// TIA Portal project "ConveyorBelt (extra)" (V13)

(* hardware
DEVICE "S7300/ET200M-Station_1"  S7-300 station
   slot 0: "Profilschiene_0"  Rail  6ES7 390-1***0-0AA0
   slot 1: "PS 307 5A_1"  PS 307 5A  6ES7 307-1EA00-0AA0
   slot 2: "SIMATIC S7-300"  CPU 314C-2 PN/DP  6ES7 314-6EH04-0AB0  V3.3
      slot 2: "PROFINET-Schnittstelle_1"  PN-IO
         slot 1: "Port_1"  Port
         slot 2: "Port_2"  Port
      slot 5: "DI 24/DO 16_1"  DI24/DO16
      slot 6: "AI 5/AO 2_1"  AI5/AO2
      slot 7: "Zählen_1"  Counter
      slot 8: "Positionieren_1"  Positioning
*)

// ===== PLC "SIMATIC S7-300"  CPU 314C-2 PN/DP =====

VAR_GLOBAL   // PLC tag table "Standard-Variablentabelle"
   "Ix_1S1" AT %I124.0 : Bool;   // Start-Taster (NO)
   "Ix_2S1" AT %I124.1 : Bool;   // Halt-Taster (NC)
   "Ix_3S1" AT %I124.2 : Bool;   // Richten-Taster (NO)
   "Ix_1B1" AT %I124.3 : Bool;   // Werkstück in Werkstückaufnahme (Ausgangsposition)
   "Ix_2B1" AT %I124.4 : Bool;   // Schwenkarm 1, Position Förderband
   "Ix_2B2" AT %I124.5 : Bool;   // Schwenkarm 1, Position Werkstückaufnahme
   "Ix_3B1" AT %I124.6 : Bool;   // Werkstück am Förderbandende
   "Ix_4B1" AT %I124.7 : Bool;   // Hubeinrichtung, Position oben
   "Ix_5B1" AT %I125.1 : Bool;   // Schwenkarm 2, Position Förderband
   "Ix_5B2" AT %I125.2 : Bool;   // Schwenkarm 2, Position Schlitten
   "Ix_6B1" AT %I125.3 : Bool;   // Werkstück in Werkstückaufnahme des Schlittens
   "Ix_7B2" AT %I125.4 : Bool;   // Schlitten, Position Werkstückaufnahme
   "Ix_7B1" AT %I125.5 : Bool;   // Schlitten, Position Werkstückübergabe
   "Ix_8B1" AT %I125.6 : Bool;   // Schwenkarm 3, Position Rollenband
   "Ix_8B2" AT %I125.7 : Bool;   // Schwenkarm 3, Position Schlitten
   "Ix_9B1" AT %I126.0 : Bool;   // Vakuum Greifer 1 eingeschaltet
   "Ix_9B2" AT %I126.1 : Bool;   // Vakuum Greifer 2 eingeschaltet
   "Ix_4B2" AT %I125.0 : Bool;   // Hubeinrichtung, Position unten
   "Ix_9B3" AT %I126.2 : Bool;   // Vakuum Greifer 3 eingeschaltet
   "Qx_1M1" AT %Q124.0 : Bool;   // Schwenkarm 1 zum Transportgut
   "Qx_2M1" AT %Q124.1 : Bool;   // Förderbandantrieb Schub 1 (NC)
   "Qx_2M2" AT %Q124.2 : Bool;   // Förderbandantrieb Schub 2 (NO)
   "Qx_3M1" AT %Q124.3 : Bool;   // Hubeinrichtung nach unten
   "Qx_4M1" AT %Q124.4 : Bool;   // Schwenkarm 2 vom Förderband zum Schlitten
   "Qx_5M1" AT %Q124.5 : Bool;   // Schlitten zum Schwenkarm 2
   "Qx_6M1" AT %Q124.6 : Bool;   // Schwenkarm 3 von der Rollenbahn zum Schlitten
   "Qx_7M1" AT %Q125.2 : Bool;   // Greifer 1 einschalten
   "Qx_7M2" AT %Q124.7 : Bool;   // Greifer 1 ausschalten
   "Qx_7M3" AT %Q125.3 : Bool;   // Greifer 2 einschalten
   "Qx_7M4" AT %Q125.0 : Bool;   // Greifer 2 ausschalten
   "Qx_7M5" AT %Q125.4 : Bool;   // Greifer 3 einschalten
   "Qx_7M6" AT %Q125.1 : Bool;   // Greifer 3 ausschalten
   "Qx_PStart" AT %Q125.5 : Bool;   // Startlampe (grün)
   "Qx_PHalt" AT %Q125.6 : Bool;   // Haltlampe (rot)
   "Qx_PRichten" AT %Q125.7 : Bool;   // Richtenlampe (orange)
   "Mx_Step0" AT %M0.0 : Bool;   // Merker: Step 0
   "Mx_Step1" AT %M0.1 : Bool;   // Merker: Step 1
   "Mx_Step2" AT %M0.2 : Bool;   // Merker: Step 2
   "Mx_Step3" AT %M0.3 : Bool;   // Merker: Step 3
   "Mx_Step4" AT %M0.4 : Bool;   // Merker: Step 4
   "Mx_Step5" AT %M0.5 : Bool;   // Merker: Step 5
   "Mx_Step6a" AT %M0.6 : Bool;   // Merker: Step 6a
   "Mx_Step7" AT %M0.7 : Bool;   // Merker: Step 7
   "Mx_Step8" AT %M1.0 : Bool;   // Merker: Step 8
   "Mx_Step9" AT %M1.1 : Bool;   // Merker: Step 9
   "Mx_Step10" AT %M1.2 : Bool;   // Merker: Step 10
   "Mx_Step11" AT %M1.3 : Bool;   // Merker: Step 11
   "Mx_Step12" AT %M1.4 : Bool;   // Merker: Step 12
   "Mx_Step13" AT %M1.5 : Bool;   // Merker: Step 13
   "Mx_Step14" AT %M1.6 : Bool;   // Merker: Step 14
   "Mx_Step15" AT %M1.7 : Bool;   // Merker: Step 15
   "Mx_Step16" AT %M2.0 : Bool;   // Merker: Step 16
   "Mx_Step17" AT %M2.1 : Bool;   // Merker: Step 17
   "Mx_Step18" AT %M2.2 : Bool;   // Merker: Step 18
   "Mx_Step19" AT %M2.3 : Bool;   // Merker: Step 19
   "Mx_Step20" AT %M2.4 : Bool;   // Merker: Step 20
   "Mx_Step21" AT %M2.5 : Bool;   // Merker: Step 21
   "Mx_Step22" AT %M2.6 : Bool;   // Merker: Step 22
   "Mx_Step23" AT %M2.7 : Bool;   // Merker: Step 23
   "MD0" AT %MD0 : DWord;   // Merker Doppel Wort 0
   "Mx_InitialFlag" AT %M3.0 : Bool;   // Merker: Initialisierung
   "Mx_Ausgangstellung" AT %M10.0 : Bool;   // Merker: Ausgangstellung
   "Mx_InitSchwenkarm1" AT %M10.1 : Bool;   // Merker: Initalisierung Schwenkarm 1
   "Mx_InitSchwenkarm2" AT %M10.2 : Bool;
   "Mx_InitHubeinrichtung" AT %M10.3 : Bool;
   "Mx_InitSchwenkarm3" AT %M10.4 : Bool;
   "Mx_InitGreifer1" AT %M10.5 : Bool;
   "Mx_InitGreifer2" AT %M10.6 : Bool;
   "Mx_InitGreifer3" AT %M10.7 : Bool;
   "MD10" AT %MD10 : DWord;
   "Mx_ResetOK" AT %M11.0 : Bool;
   "Mx_FStart" AT %M11.1 : Bool;
   "Mx_Step6b" AT %M11.2 : Bool;   // Merker: Step 6b
   "Mb10" AT %MB10 : Byte;   // Merkerbyte10
END_VAR

DATA_BLOCK "Ausgangsstellung_DB"   // DB2
{ S7_Optimized_Access := 'FALSE' }
VERSION : 0.1
// stored: InstanceOfName Ausgangsstellung
"Ausgangsstellung"
BEGIN
END_DATA_BLOCK

FUNCTION_BLOCK "Ausgangsstellung"   // FB1, FBD
{ S7_Optimized_Access := 'FALSE' }
VERSION : 0.1
BEGIN

REGION Network 1: Schwnkarm 1 zum Förderband
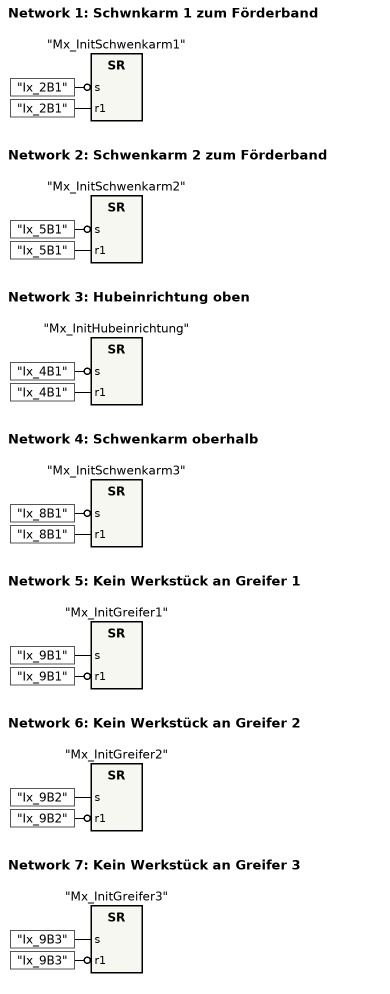
   IF NOT "Ix_2B1" THEN
       "Mx_InitSchwenkarm1" := TRUE;   // SR flip-flop
   END_IF;
   IF "Ix_2B1" THEN "Mx_InitSchwenkarm1" := FALSE; END_IF;
END_REGION

REGION Network 2: Schwenkarm 2 zum Förderband
   IF NOT "Ix_5B1" THEN
       "Mx_InitSchwenkarm2" := TRUE;   // SR flip-flop
   END_IF;
   IF "Ix_5B1" THEN "Mx_InitSchwenkarm2" := FALSE; END_IF;
END_REGION

REGION Network 3: Hubeinrichtung oben
   IF NOT "Ix_4B1" THEN
       "Mx_InitHubeinrichtung" := TRUE;   // SR flip-flop
   END_IF;
   IF "Ix_4B1" THEN "Mx_InitHubeinrichtung" := FALSE; END_IF;
END_REGION

REGION Network 4: Schwenkarm oberhalb
   IF NOT "Ix_8B1" THEN
       "Mx_InitSchwenkarm3" := TRUE;   // SR flip-flop
   END_IF;
   IF "Ix_8B1" THEN "Mx_InitSchwenkarm3" := FALSE; END_IF;
END_REGION

REGION Network 5: Kein Werkstück an Greifer 1
   IF "Ix_9B1" THEN
       "Mx_InitGreifer1" := TRUE;   // SR flip-flop
   END_IF;
   IF NOT "Ix_9B1" THEN "Mx_InitGreifer1" := FALSE; END_IF;
END_REGION

REGION Network 6: Kein Werkstück an Greifer 2
   IF "Ix_9B2" THEN
       "Mx_InitGreifer2" := TRUE;   // SR flip-flop
   END_IF;
   IF NOT "Ix_9B2" THEN "Mx_InitGreifer2" := FALSE; END_IF;
END_REGION

REGION Network 7: Kein Werkstück an Greifer 3
   IF "Ix_9B3" THEN
       "Mx_InitGreifer3" := TRUE;   // SR flip-flop
   END_IF;
   IF NOT "Ix_9B3" THEN "Mx_InitGreifer3" := FALSE; END_IF;
END_REGION
END_FUNCTION_BLOCK

FUNCTION "FC1 Grafcet" : Void   // FC1, FBD
{ S7_Optimized_Access := 'FALSE' }
VERSION : 0.1
BEGIN

REGION Network 1: Step 1
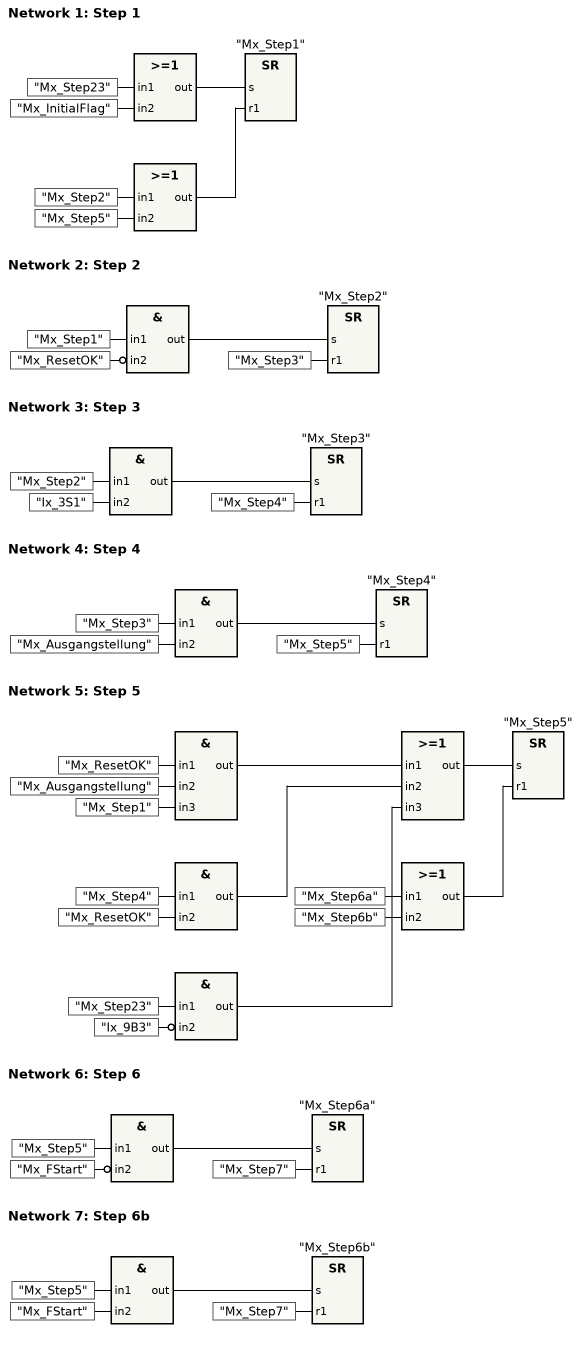
   IF "Mx_Step23" OR "Mx_InitialFlag" THEN
       "Mx_Step1" := TRUE;   // SR flip-flop
   END_IF;
   IF "Mx_Step2" OR "Mx_Step5" THEN "Mx_Step1" := FALSE; END_IF;
END_REGION

REGION Network 2: Step 2
   IF "Mx_Step1" AND NOT "Mx_ResetOK" THEN
       "Mx_Step2" := TRUE;   // SR flip-flop
   END_IF;
   IF "Mx_Step3" THEN "Mx_Step2" := FALSE; END_IF;
END_REGION

REGION Network 3: Step 3
   IF "Mx_Step2" AND "Ix_3S1" THEN
       "Mx_Step3" := TRUE;   // SR flip-flop
   END_IF;
   IF "Mx_Step4" THEN "Mx_Step3" := FALSE; END_IF;
END_REGION

REGION Network 4: Step 4
   IF "Mx_Step3" AND "Mx_Ausgangstellung" THEN
       "Mx_Step4" := TRUE;   // SR flip-flop
   END_IF;
   IF "Mx_Step5" THEN "Mx_Step4" := FALSE; END_IF;
END_REGION

REGION Network 5: Step 5
   IF ("Mx_ResetOK" AND "Mx_Ausgangstellung" AND "Mx_Step1") OR ("Mx_Step4" AND "Mx_ResetOK") OR ("Mx_Step23" AND NOT "Ix_9B3") THEN
       "Mx_Step5" := TRUE;   // SR flip-flop
   END_IF;
   IF "Mx_Step6a" OR "Mx_Step6b" THEN "Mx_Step5" := FALSE; END_IF;
END_REGION

REGION Network 6: Step 6
   IF "Mx_Step5" AND NOT "Mx_FStart" THEN
       "Mx_Step6a" := TRUE;   // SR flip-flop
   END_IF;
   IF "Mx_Step7" THEN "Mx_Step6a" := FALSE; END_IF;
END_REGION

REGION Network 7: Step 6b
   IF "Mx_Step5" AND "Mx_FStart" THEN
       "Mx_Step6b" := TRUE;   // SR flip-flop
   END_IF;
   IF "Mx_Step7" THEN "Mx_Step6b" := FALSE; END_IF;
END_REGION

REGION Network 8: Step 7
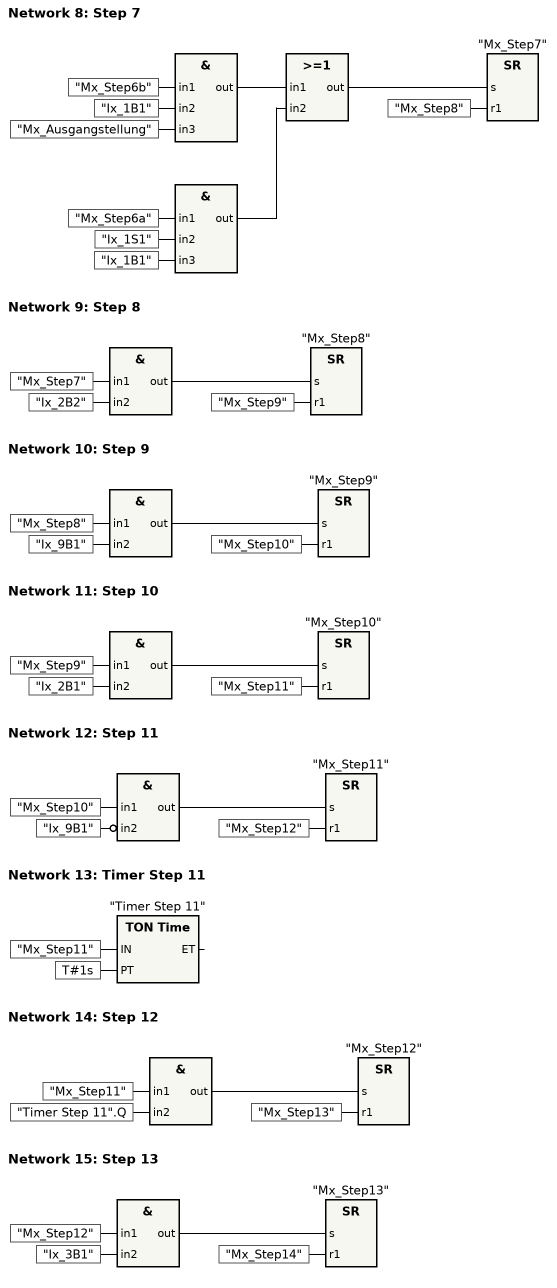
   IF ("Mx_Step6b" AND "Ix_1B1" AND "Mx_Ausgangstellung") OR ("Mx_Step6a" AND "Ix_1S1" AND "Ix_1B1") THEN
       "Mx_Step7" := TRUE;   // SR flip-flop
   END_IF;
   IF "Mx_Step8" THEN "Mx_Step7" := FALSE; END_IF;
END_REGION

REGION Network 9: Step 8
   IF "Mx_Step7" AND "Ix_2B2" THEN
       "Mx_Step8" := TRUE;   // SR flip-flop
   END_IF;
   IF "Mx_Step9" THEN "Mx_Step8" := FALSE; END_IF;
END_REGION

REGION Network 10: Step 9
   IF "Mx_Step8" AND "Ix_9B1" THEN
       "Mx_Step9" := TRUE;   // SR flip-flop
   END_IF;
   IF "Mx_Step10" THEN "Mx_Step9" := FALSE; END_IF;
END_REGION

REGION Network 11: Step 10
   IF "Mx_Step9" AND "Ix_2B1" THEN
       "Mx_Step10" := TRUE;   // SR flip-flop
   END_IF;
   IF "Mx_Step11" THEN "Mx_Step10" := FALSE; END_IF;
END_REGION

REGION Network 12: Step 11
   IF "Mx_Step10" AND NOT "Ix_9B1" THEN
       "Mx_Step11" := TRUE;   // SR flip-flop
   END_IF;
   IF "Mx_Step12" THEN "Mx_Step11" := FALSE; END_IF;
END_REGION

REGION Network 13: Timer Step 11
   "Timer Step 11".TON(IN := "Mx_Step11", PT := T#1s);
END_REGION

REGION Network 14: Step 12
   IF "Mx_Step11" AND "Timer Step 11".Q THEN
       "Mx_Step12" := TRUE;   // SR flip-flop
   END_IF;
   IF "Mx_Step13" THEN "Mx_Step12" := FALSE; END_IF;
END_REGION

REGION Network 15: Step 13
   IF "Mx_Step12" AND "Ix_3B1" THEN
       "Mx_Step13" := TRUE;   // SR flip-flop
   END_IF;
   IF "Mx_Step14" THEN "Mx_Step13" := FALSE; END_IF;
END_REGION

REGION Network 16: Step 14
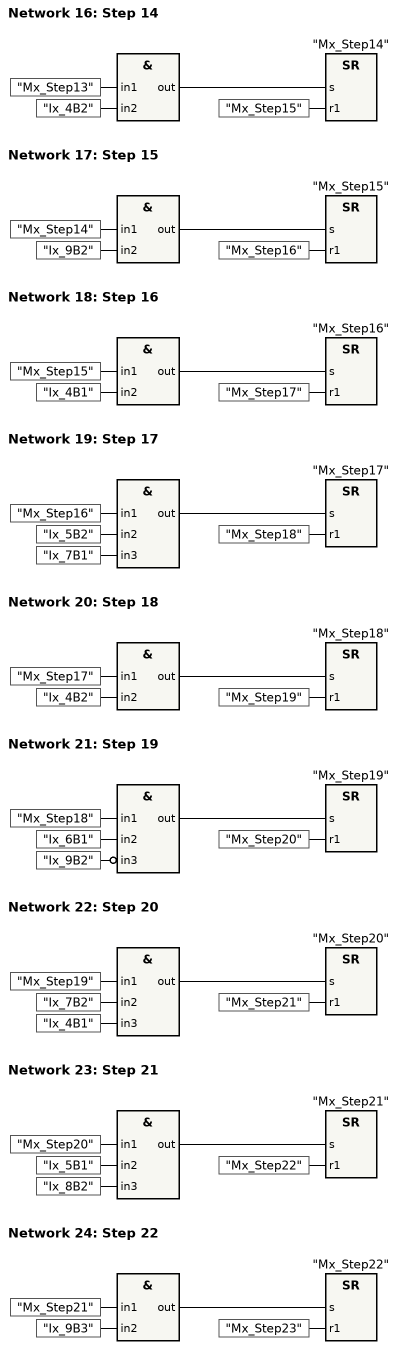
   IF "Mx_Step13" AND "Ix_4B2" THEN
       "Mx_Step14" := TRUE;   // SR flip-flop
   END_IF;
   IF "Mx_Step15" THEN "Mx_Step14" := FALSE; END_IF;
END_REGION

REGION Network 17: Step 15
   IF "Mx_Step14" AND "Ix_9B2" THEN
       "Mx_Step15" := TRUE;   // SR flip-flop
   END_IF;
   IF "Mx_Step16" THEN "Mx_Step15" := FALSE; END_IF;
END_REGION

REGION Network 18: Step 16
   IF "Mx_Step15" AND "Ix_4B1" THEN
       "Mx_Step16" := TRUE;   // SR flip-flop
   END_IF;
   IF "Mx_Step17" THEN "Mx_Step16" := FALSE; END_IF;
END_REGION

REGION Network 19: Step 17
   IF "Mx_Step16" AND "Ix_5B2" AND "Ix_7B1" THEN
       "Mx_Step17" := TRUE;   // SR flip-flop
   END_IF;
   IF "Mx_Step18" THEN "Mx_Step17" := FALSE; END_IF;
END_REGION

REGION Network 20: Step 18
   IF "Mx_Step17" AND "Ix_4B2" THEN
       "Mx_Step18" := TRUE;   // SR flip-flop
   END_IF;
   IF "Mx_Step19" THEN "Mx_Step18" := FALSE; END_IF;
END_REGION

REGION Network 21: Step 19
   IF "Mx_Step18" AND "Ix_6B1" AND NOT "Ix_9B2" THEN
       "Mx_Step19" := TRUE;   // SR flip-flop
   END_IF;
   IF "Mx_Step20" THEN "Mx_Step19" := FALSE; END_IF;
END_REGION

REGION Network 22: Step 20
   IF "Mx_Step19" AND "Ix_7B2" AND "Ix_4B1" THEN
       "Mx_Step20" := TRUE;   // SR flip-flop
   END_IF;
   IF "Mx_Step21" THEN "Mx_Step20" := FALSE; END_IF;
END_REGION

REGION Network 23: Step 21
   IF "Mx_Step20" AND "Ix_5B1" AND "Ix_8B2" THEN
       "Mx_Step21" := TRUE;   // SR flip-flop
   END_IF;
   IF "Mx_Step22" THEN "Mx_Step21" := FALSE; END_IF;
END_REGION

REGION Network 24: Step 22
   IF "Mx_Step21" AND "Ix_9B3" THEN
       "Mx_Step22" := TRUE;   // SR flip-flop
   END_IF;
   IF "Mx_Step23" THEN "Mx_Step22" := FALSE; END_IF;
END_REGION

REGION Network 25: Step 23
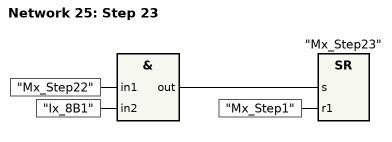
   IF "Mx_Step22" AND "Ix_8B1" THEN
       "Mx_Step23" := TRUE;   // SR flip-flop
   END_IF;
   IF "Mx_Step1" THEN "Mx_Step23" := FALSE; END_IF;
END_REGION
END_FUNCTION

FUNCTION "FC Actions" : Void   // FC2, FBD
{ S7_Optimized_Access := 'FALSE' }
VERSION : 0.1
BEGIN

REGION Network 2: Lampe Richten P_R
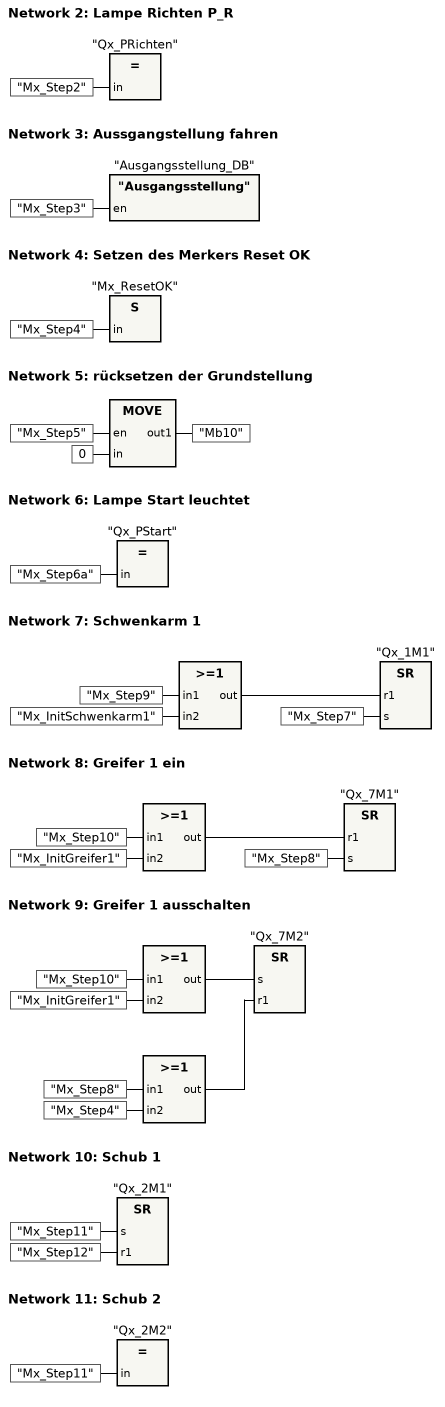
   "Qx_PRichten" := "Mx_Step2";
END_REGION

REGION Network 3: Aussgangstellung fahren
   IF "Mx_Step3" THEN
       "Ausgangsstellung_DB"();   // "Ausgangsstellung"
   END_IF;
END_REGION

REGION Network 4: Setzen des Merkers Reset OK
   IF "Mx_Step4" THEN "Mx_ResetOK" := TRUE; END_IF;
END_REGION

REGION Network 5: rücksetzen der Grundstellung
   IF "Mx_Step5" THEN "Mb10" := 0; END_IF;
END_REGION

REGION Network 6: Lampe Start leuchtet
   "Qx_PStart" := "Mx_Step6a";
END_REGION

REGION Network 7: Schwenkarm 1
   IF "Mx_Step7" THEN
       "Qx_1M1" := TRUE;   // SR flip-flop
   END_IF;
   IF "Mx_Step9" OR "Mx_InitSchwenkarm1" THEN "Qx_1M1" := FALSE; END_IF;
END_REGION

REGION Network 8: Greifer 1 ein
   IF "Mx_Step8" THEN
       "Qx_7M1" := TRUE;   // SR flip-flop
   END_IF;
   IF "Mx_Step10" OR "Mx_InitGreifer1" THEN "Qx_7M1" := FALSE; END_IF;
END_REGION

REGION Network 9: Greifer 1 ausschalten
   IF "Mx_Step10" OR "Mx_InitGreifer1" THEN
       "Qx_7M2" := TRUE;   // SR flip-flop
   END_IF;
   IF "Mx_Step8" OR "Mx_Step4" THEN "Qx_7M2" := FALSE; END_IF;
END_REGION

REGION Network 10: Schub 1
   IF "Mx_Step11" THEN
       "Qx_2M1" := TRUE;   // SR flip-flop
   END_IF;
   IF "Mx_Step12" THEN "Qx_2M1" := FALSE; END_IF;
END_REGION

REGION Network 11: Schub 2
   "Qx_2M2" := "Mx_Step11";
END_REGION

REGION Network 12: Hubeinrichtung
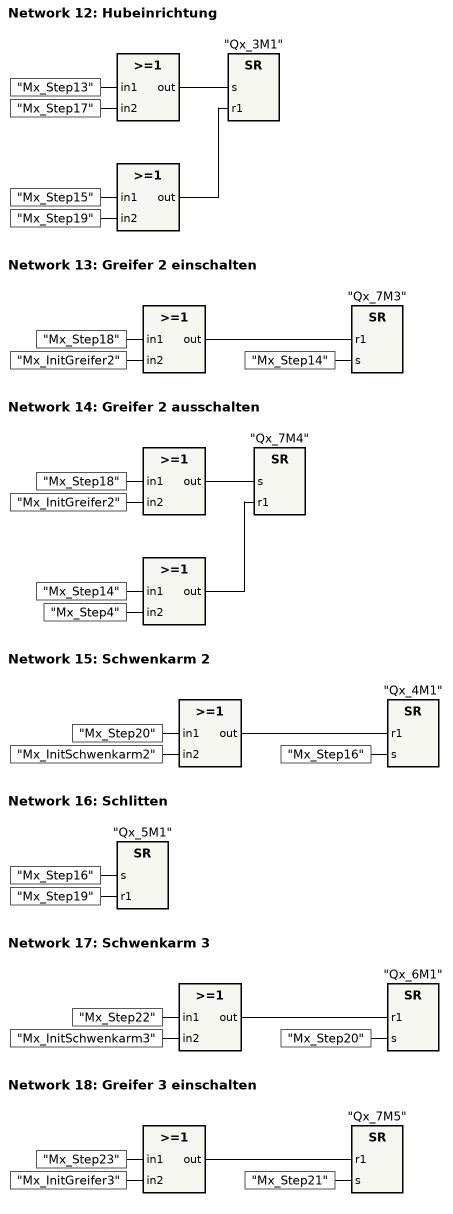
   IF "Mx_Step13" OR "Mx_Step17" THEN
       "Qx_3M1" := TRUE;   // SR flip-flop
   END_IF;
   IF "Mx_Step15" OR "Mx_Step19" THEN "Qx_3M1" := FALSE; END_IF;
END_REGION

REGION Network 13: Greifer 2 einschalten
   IF "Mx_Step14" THEN
       "Qx_7M3" := TRUE;   // SR flip-flop
   END_IF;
   IF "Mx_Step18" OR "Mx_InitGreifer2" THEN "Qx_7M3" := FALSE; END_IF;
END_REGION

REGION Network 14: Greifer 2 ausschalten
   IF "Mx_Step18" OR "Mx_InitGreifer2" THEN
       "Qx_7M4" := TRUE;   // SR flip-flop
   END_IF;
   IF "Mx_Step14" OR "Mx_Step4" THEN "Qx_7M4" := FALSE; END_IF;
END_REGION

REGION Network 15: Schwenkarm 2
   IF "Mx_Step16" THEN
       "Qx_4M1" := TRUE;   // SR flip-flop
   END_IF;
   IF "Mx_Step20" OR "Mx_InitSchwenkarm2" THEN "Qx_4M1" := FALSE; END_IF;
END_REGION

REGION Network 16: Schlitten
   IF "Mx_Step16" THEN
       "Qx_5M1" := TRUE;   // SR flip-flop
   END_IF;
   IF "Mx_Step19" THEN "Qx_5M1" := FALSE; END_IF;
END_REGION

REGION Network 17: Schwenkarm 3
   IF "Mx_Step20" THEN
       "Qx_6M1" := TRUE;   // SR flip-flop
   END_IF;
   IF "Mx_Step22" OR "Mx_InitSchwenkarm3" THEN "Qx_6M1" := FALSE; END_IF;
END_REGION

REGION Network 18: Greifer 3 einschalten
   IF "Mx_Step21" THEN
       "Qx_7M5" := TRUE;   // SR flip-flop
   END_IF;
   IF "Mx_Step23" OR "Mx_InitGreifer3" THEN "Qx_7M5" := FALSE; END_IF;
END_REGION

REGION Network 19: Greifer 3 ausschalten
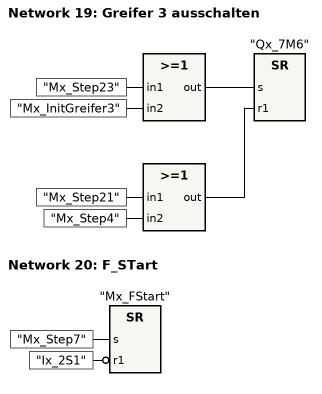
   IF "Mx_Step23" OR "Mx_InitGreifer3" THEN
       "Qx_7M6" := TRUE;   // SR flip-flop
   END_IF;
   IF "Mx_Step21" OR "Mx_Step4" THEN "Qx_7M6" := FALSE; END_IF;
END_REGION

REGION Network 20: F_STart
   IF "Mx_Step7" THEN
       "Mx_FStart" := TRUE;   // SR flip-flop
   END_IF;
   IF NOT "Ix_2S1" THEN "Mx_FStart" := FALSE; END_IF;
END_REGION
END_FUNCTION

ORGANIZATION_BLOCK "Main"   // OB1, FBD
TITLE = "Main Program Sweep (Cycle)"
{ S7_Optimized_Access := 'FALSE' }
VERSION : 0.1
BEGIN

REGION Network 1
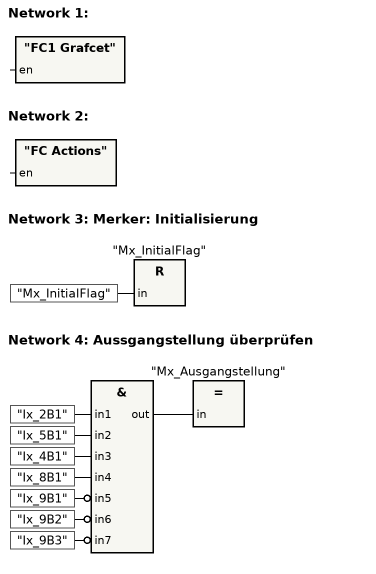
   "FC1 Grafcet"();
END_REGION

REGION Network 2
   "FC Actions"();
END_REGION

REGION Network 3: Merker: Initialisierung
   IF "Mx_InitialFlag" THEN "Mx_InitialFlag" := FALSE; END_IF;
END_REGION

REGION Network 4: Aussgangstellung überprüfen
   "Mx_Ausgangstellung" := "Ix_2B1" AND "Ix_5B1" AND "Ix_4B1" AND "Ix_8B1" AND NOT "Ix_9B1" AND NOT "Ix_9B2" AND NOT "Ix_9B3";
END_REGION
END_ORGANIZATION_BLOCK

ORGANIZATION_BLOCK "COMPLETE RESTART"   // OB100, FBD
TITLE = "Complete Restart"
{ S7_Optimized_Access := 'FALSE' }
VERSION : 0.1
BEGIN

REGION Network 1: Resset all Doubelword 0
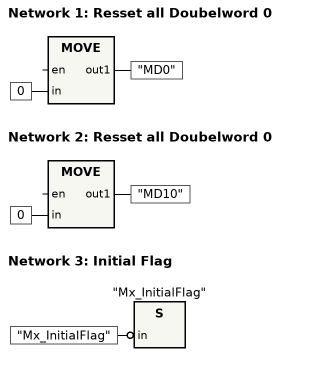
   "MD0" := 0;
END_REGION

REGION Network 2: Resset all Doubelword 0
   "MD10" := 0;
END_REGION

REGION Network 3: Initial Flag
   IF NOT "Mx_InitialFlag" THEN "Mx_InitialFlag" := TRUE; END_IF;
END_REGION
END_ORGANIZATION_BLOCK